{attribute addProperty BoxType "EL3311-0000-0018"}
{attribute addProperty Id "StatusAT %I*Status_34730D861621ValueAT %I*INT16217"}
{attribute addProperty CRC "4291910102"}
{attribute addProperty SizeInBites "32"}
{attribute addProperty SizeInBytes "4"}
TYPE TC_Inputs_FFD159D6 :
STRUCT
	{attribute addProperty Name "Status"}
	Status AT %I* : Status_34730D86;
	{attribute addProperty Name "Value"}
	Value AT %I* : INT;
END_STRUCT
END_TYPE

(* stored: Version 1.2.0.0, ProductVersion 3.1.4024.9
   DUT TC_Inputs_FFD159D6: Id {bf86b364-81e5-4ba5-8a7a-115dc70493d2} *)
